// TIA Portal project "Automated Ware house" (V14)
// Vorlageprojekt für das Buch mit Zielsystem S7-1200

(* hardware
DEVICE "S7-1200-Station_1"  S7-1200 Station
   slot 0: "Baugruppenträger_0"  Rack  V1.0
   slot 1: "PLC_1"  CPU 1211C DC/DC/DC  6ES7 211-1AE40-0XB0  V4.1
*)

// ===== PLC "PLC_1"  CPU 1211C DC/DC/DC =====

VAR_GLOBAL   // PLC tag table "Standard-Variablentabelle"
   "At entry" AT %I0.0 : Bool;
   "at load" AT %I0.1 : Bool;
   "at left" AT %I0.2 : Bool;
   "at middle" AT %I0.3 : Bool;
   "at right" AT %I0.4 : Bool;
   "at unload" AT %I0.5 : Bool;
   "at exit" AT %I0.6 : Bool;
   "moving x" AT %I0.7 : Bool;
   "moving z" AT %I1.0 : Bool;
   "start" AT %I1.1 : Bool;
   "reset" AT %I1.2 : Bool;
   "stop" AT %I1.3 : Bool;
   "emergency stop" AT %I1.4 : Bool;
   "auto" AT %I1.5 : Bool;
   "entry conveyor" AT %Q0.0 : Bool;
   "load conveyor" AT %Q0.1 : Bool;
   "forks left" AT %Q0.2 : Bool;
   "fork right" AT %Q0.3 : Bool;
   "lift" AT %Q0.4 : Bool;
   "unload conveyor" AT %Q0.5 : Bool;
   "exit conveyor" AT %Q0.6 : Bool;
   "start light" AT %Q0.7 : Bool;
   "reset light" AT %Q1.0 : Bool;
   "stop light" AT %Q1.1 : Bool;
   "target position" AT %QD30 : DInt;
   "Tag_1" AT %M20.0 : Bool;
   "Tag_2" AT %M20.1 : Bool;
   "Tag_4" AT %MD4 : DInt;
   "Tag_7" AT %MD12 : DInt;
   "Tag_8" AT %M20.2 : Bool;
   "Tag_3" AT %M20.3 : Bool;
   "Tag_14" AT %M21.2 : Bool;
   "Tag_16" AT %M21.4 : Bool;
   "Tag_18" AT %MD8 : DInt;
   "Tag_6" AT %M21.6 : Bool;
   "Tag_19" AT %M21.7 : Bool;
   "Tag_20" AT %M22.1 : Bool;
   "Tag_22" AT %M22.3 : Bool;
   "Tag_5" AT %M22.2 : Bool;
END_VAR

// folder: System blocks/Program resources

DATA_BLOCK "IEC_Counter_0_DB"   // DB1
{ S7_Optimized_Access := 'TRUE' }
AUTHOR : Simatic
FAMILY : IEC
NAME : CNTR
VERSION : 1.0
// stored: InstanceOfName IEC_COUNTER
"IEC_COUNTER"
BEGIN
END_DATA_BLOCK

DATA_BLOCK "IEC_Timer_0_DB"   // DB2
{ S7_Optimized_Access := 'TRUE' }
AUTHOR : Simatic
FAMILY : IEC
NAME : IEC_TMR
VERSION : 1.0
// stored: InstanceOfName IEC_TIMER
"IEC_TIMER"
BEGIN
END_DATA_BLOCK

// folder: (top level)

FUNCTION "Conveyors" : Void   // FC1, LAD
{ S7_Optimized_Access := 'TRUE' }
VERSION : 0.1
   VAR_TEMP   // added for the SCL form of the ladder/FBD networks
      _w1 : Bool;
   END_VAR
BEGIN

REGION Network 1
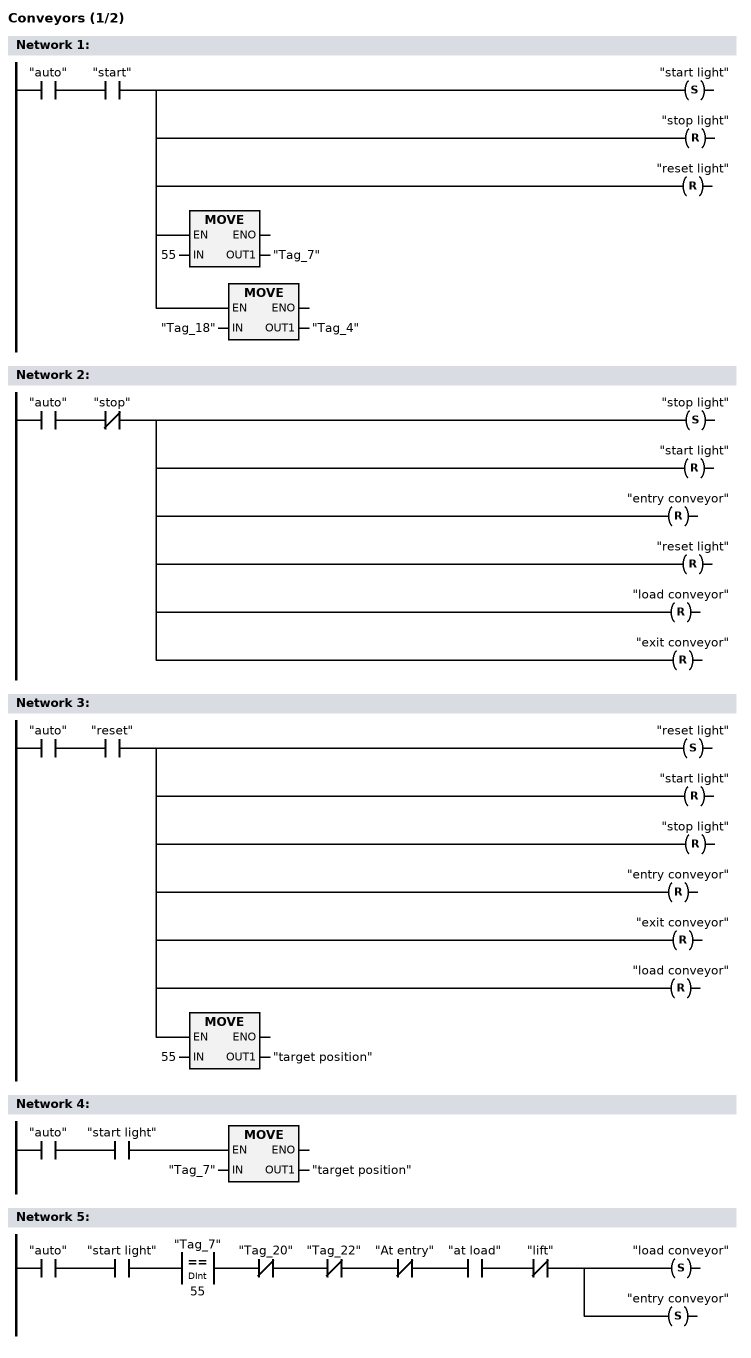
   RUNG wire#powerrail
      Contact( "auto" )
      Contact( "start" )
      wire#w1
      S_Coil( "start light" )
   END_RUNG
   RUNG wire#w1
      R_Coil( "stop light" )
   END_RUNG
   RUNG wire#w1
      R_Coil( "reset light" )
   END_RUNG
   RUNG wire#w1
      Move(in := 55, out1 => "Tag_7")
   END_RUNG
   RUNG wire#w1
      Move(in := "Tag_18", out1 => "Tag_4")
   END_RUNG
   // the same network as SCL:
   IF "auto" AND "start" THEN
       "start light" := TRUE;
       "stop light" := FALSE;
       "reset light" := FALSE;
       "Tag_7" := 55;
       "Tag_4" := "Tag_18";
   END_IF;
END_REGION

REGION Network 2
   RUNG wire#powerrail
      Contact( "auto" )
      I_Contact( "stop" )
      wire#w1
      S_Coil( "stop light" )
   END_RUNG
   RUNG wire#w1
      R_Coil( "start light" )
   END_RUNG
   RUNG wire#w1
      R_Coil( "entry conveyor" )
   END_RUNG
   RUNG wire#w1
      R_Coil( "reset light" )
   END_RUNG
   RUNG wire#w1
      R_Coil( "load conveyor" )
   END_RUNG
   RUNG wire#w1
      R_Coil( "exit conveyor" )
   END_RUNG
   // the same network as SCL:
   IF "auto" AND NOT "stop" THEN
       "stop light" := TRUE;
       "start light" := FALSE;
       "entry conveyor" := FALSE;
       "reset light" := FALSE;
       "load conveyor" := FALSE;
       "exit conveyor" := FALSE;
   END_IF;
END_REGION

REGION Network 3
   RUNG wire#powerrail
      Contact( "auto" )
      Contact( "reset" )
      wire#w1
      S_Coil( "reset light" )
   END_RUNG
   RUNG wire#w1
      R_Coil( "start light" )
   END_RUNG
   RUNG wire#w1
      R_Coil( "stop light" )
   END_RUNG
   RUNG wire#w1
      R_Coil( "entry conveyor" )
   END_RUNG
   RUNG wire#w1
      R_Coil( "exit conveyor" )
   END_RUNG
   RUNG wire#w1
      R_Coil( "load conveyor" )
   END_RUNG
   RUNG wire#w1
      Move(in := 55, out1 => "target position")
   END_RUNG
   // the same network as SCL:
   IF "auto" AND "reset" THEN
       "reset light" := TRUE;
       "start light" := FALSE;
       "stop light" := FALSE;
       "entry conveyor" := FALSE;
       "exit conveyor" := FALSE;
       "load conveyor" := FALSE;
       "target position" := 55;
   END_IF;
END_REGION

REGION Network 4
   RUNG wire#powerrail
      Contact( "auto" )
      Contact( "start light" )
      Move(in := "Tag_7", out1 => "target position")
   END_RUNG
   // the same network as SCL:
   IF "auto" AND "start light" THEN "target position" := "Tag_7"; END_IF;
END_REGION

REGION Network 5
   RUNG wire#powerrail
      Contact( "auto" )
      Contact( "start light" )
      { S7_Templates := "SrcType := DInt" } EQ_Contact(in1 := "Tag_7", in2 := 55)
      I_Contact( "Tag_20" )
      I_Contact( "Tag_22" )
      I_Contact( "At entry" )
      Contact( "at load" )
      I_Contact( "lift" )
      wire#w1
      S_Coil( "load conveyor" )
   END_RUNG
   RUNG wire#w1
      S_Coil( "entry conveyor" )
   END_RUNG
   // the same network as SCL:
   IF "auto" AND "start light" AND ("Tag_7" = 55) AND NOT "Tag_20" AND NOT "Tag_22" AND NOT "At entry" AND "at load" AND NOT "lift" THEN
       "load conveyor" := TRUE;
       "entry conveyor" := TRUE;
   END_IF;
END_REGION

REGION Network 6
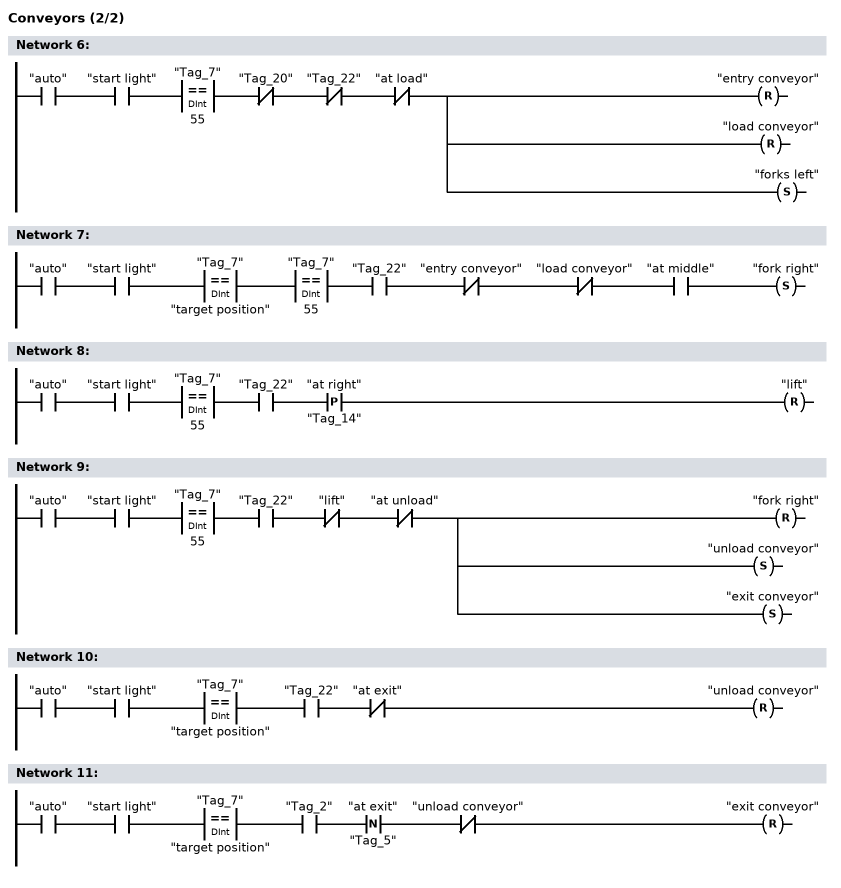
   RUNG wire#powerrail
      Contact( "auto" )
      Contact( "start light" )
      { S7_Templates := "SrcType := DInt" } EQ_Contact(in1 := "Tag_7", in2 := 55)
      I_Contact( "Tag_20" )
      I_Contact( "Tag_22" )
      I_Contact( "at load" )
      wire#w1
      R_Coil( "entry conveyor" )
   END_RUNG
   RUNG wire#w1
      R_Coil( "load conveyor" )
   END_RUNG
   RUNG wire#w1
      S_Coil( "forks left" )
   END_RUNG
   // the same network as SCL:
   IF "auto" AND "start light" AND ("Tag_7" = 55) AND NOT "Tag_20" AND NOT "Tag_22" AND NOT "at load" THEN
       "entry conveyor" := FALSE;
       "load conveyor" := FALSE;
       "forks left" := TRUE;
   END_IF;
END_REGION

REGION Network 7
   RUNG wire#powerrail
      Contact( "auto" )
      Contact( "start light" )
      { S7_Templates := "SrcType := DInt" } EQ_Contact(in1 := "Tag_7", in2 := "target position")
      { S7_Templates := "SrcType := DInt" } EQ_Contact(in1 := "Tag_7", in2 := 55)
      Contact( "Tag_22" )
      I_Contact( "entry conveyor" )
      I_Contact( "load conveyor" )
      Contact( "at middle" )
      S_Coil( "fork right" )
   END_RUNG
   // the same network as SCL:
   IF "auto" AND "start light" AND ("Tag_7" = "target position") AND ("Tag_7" = 55) AND "Tag_22" AND NOT "entry conveyor" AND NOT "load conveyor" AND "at middle" THEN
       "fork right" := TRUE;
   END_IF;
END_REGION

REGION Network 8
   RUNG wire#powerrail
      Contact( "auto" )
      Contact( "start light" )
      { S7_Templates := "SrcType := DInt" } EQ_Contact(in1 := "Tag_7", in2 := 55)
      Contact( "Tag_22" )
      P_Contact(operand := "at right", bit := "Tag_14")
      R_Coil( "lift" )
   END_RUNG
   // the same network as SCL:
   #_w1 := "auto" AND "start light" AND ("Tag_7" = 55) AND "Tag_22" AND "at right" AND NOT "Tag_14";   // rising edge of "at right"
   "Tag_14" := "at right";
   IF #_w1 THEN "lift" := FALSE; END_IF;
END_REGION

REGION Network 9
   RUNG wire#powerrail
      Contact( "auto" )
      Contact( "start light" )
      { S7_Templates := "SrcType := DInt" } EQ_Contact(in1 := "Tag_7", in2 := 55)
      Contact( "Tag_22" )
      I_Contact( "lift" )
      I_Contact( "at unload" )
      wire#w1
      R_Coil( "fork right" )
   END_RUNG
   RUNG wire#w1
      S_Coil( "unload conveyor" )
   END_RUNG
   RUNG wire#w1
      S_Coil( "exit conveyor" )
   END_RUNG
   // the same network as SCL:
   IF "auto" AND "start light" AND ("Tag_7" = 55) AND "Tag_22" AND NOT "lift" AND NOT "at unload" THEN
       "fork right" := FALSE;
       "unload conveyor" := TRUE;
       "exit conveyor" := TRUE;
   END_IF;
END_REGION

REGION Network 10
   RUNG wire#powerrail
      Contact( "auto" )
      Contact( "start light" )
      { S7_Templates := "SrcType := DInt" } EQ_Contact(in1 := "Tag_7", in2 := "target position")
      Contact( "Tag_22" )
      I_Contact( "at exit" )
      R_Coil( "unload conveyor" )
   END_RUNG
   // the same network as SCL:
   IF "auto" AND "start light" AND ("Tag_7" = "target position") AND "Tag_22" AND NOT "at exit" THEN
       "unload conveyor" := FALSE;
   END_IF;
END_REGION

REGION Network 11
   RUNG wire#powerrail
      Contact( "auto" )
      Contact( "start light" )
      { S7_Templates := "SrcType := DInt" } EQ_Contact(in1 := "Tag_7", in2 := "target position")
      Contact( "Tag_2" )
      N_Contact(operand := "at exit", bit := "Tag_5")
      I_Contact( "unload conveyor" )
      R_Coil( "exit conveyor" )
   END_RUNG
   // the same network as SCL:
   #_w1 := "auto" AND "start light" AND ("Tag_7" = "target position") AND "Tag_2" AND NOT "at exit" AND "Tag_5";   // falling edge of "at exit"
   "Tag_5" := "at exit";
   IF #_w1 AND NOT "unload conveyor" THEN "exit conveyor" := FALSE; END_IF;
END_REGION
END_FUNCTION

FUNCTION "Shifting" : Void   // FC2, LAD
{ S7_Optimized_Access := 'TRUE' }
VERSION : 0.1
   VAR_TEMP   // added for the SCL form of the ladder/FBD networks
      _w1 : Bool;
   END_VAR
BEGIN

REGION Network 1
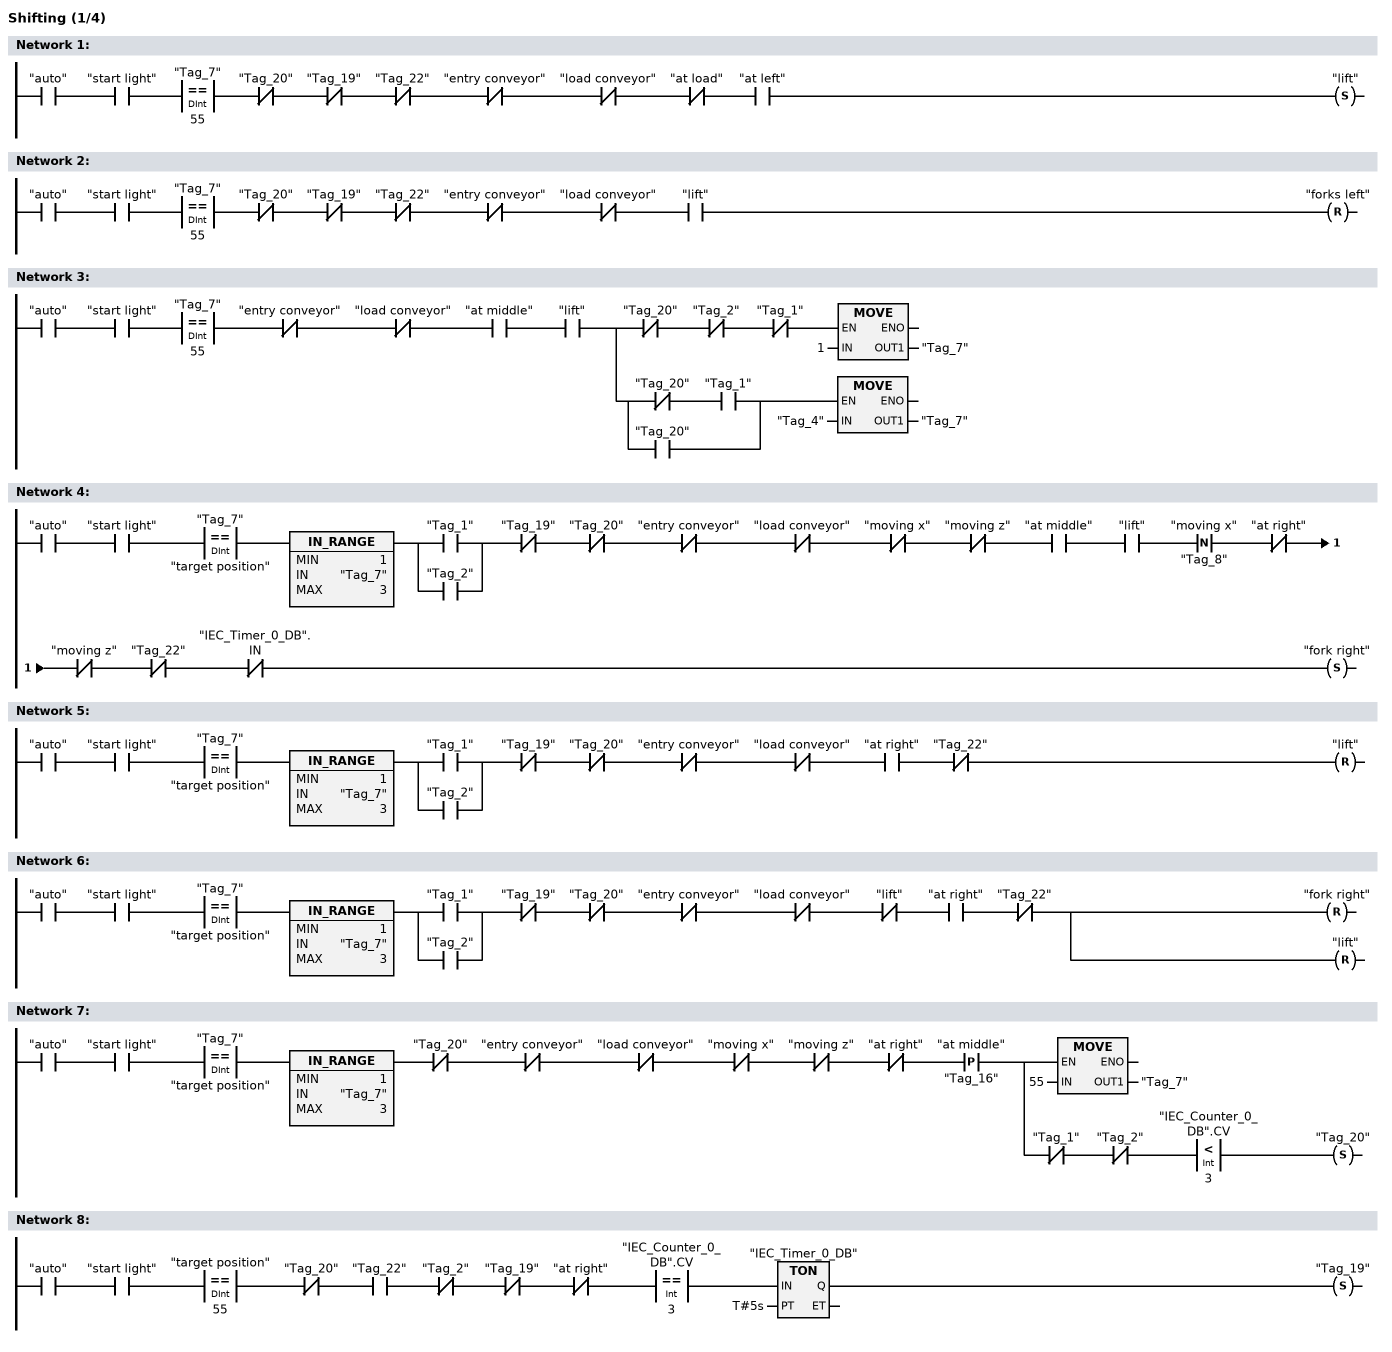
   RUNG wire#powerrail
      Contact( "auto" )
      Contact( "start light" )
      { S7_Templates := "SrcType := DInt" } EQ_Contact(in1 := "Tag_7", in2 := 55)
      I_Contact( "Tag_20" )
      I_Contact( "Tag_19" )
      I_Contact( "Tag_22" )
      I_Contact( "entry conveyor" )
      I_Contact( "load conveyor" )
      I_Contact( "at load" )
      Contact( "at left" )
      S_Coil( "lift" )
   END_RUNG
   // the same network as SCL:
   IF "auto" AND "start light" AND ("Tag_7" = 55) AND NOT "Tag_20" AND NOT "Tag_19" AND NOT "Tag_22" AND NOT "entry conveyor" AND NOT "load conveyor" AND NOT "at load" AND "at left" THEN
       "lift" := TRUE;
   END_IF;
END_REGION

REGION Network 2
   RUNG wire#powerrail
      Contact( "auto" )
      Contact( "start light" )
      { S7_Templates := "SrcType := DInt" } EQ_Contact(in1 := "Tag_7", in2 := 55)
      I_Contact( "Tag_20" )
      I_Contact( "Tag_19" )
      I_Contact( "Tag_22" )
      I_Contact( "entry conveyor" )
      I_Contact( "load conveyor" )
      Contact( "lift" )
      R_Coil( "forks left" )
   END_RUNG
   // the same network as SCL:
   IF "auto" AND "start light" AND ("Tag_7" = 55) AND NOT "Tag_20" AND NOT "Tag_19" AND NOT "Tag_22" AND NOT "entry conveyor" AND NOT "load conveyor" AND "lift" THEN
       "forks left" := FALSE;
   END_IF;
END_REGION

REGION Network 3
   RUNG wire#powerrail
      Contact( "auto" )
      Contact( "start light" )
      { S7_Templates := "SrcType := DInt" } EQ_Contact(in1 := "Tag_7", in2 := 55)
      I_Contact( "entry conveyor" )
      I_Contact( "load conveyor" )
      Contact( "at middle" )
      Contact( "lift" )
      wire#w1
      I_Contact( "Tag_20" )
      I_Contact( "Tag_2" )
      I_Contact( "Tag_1" )
      Move(in := 1, out1 => "Tag_7")
   END_RUNG
   RUNG wire#w1
      I_Contact( "Tag_20" )
      Contact( "Tag_1" )
      wire#w2
      Move(in := "Tag_4", out1 => "Tag_7")
   END_RUNG
   RUNG wire#w1
      Contact( "Tag_20" )
   END_RUNG wire#w2
   // the same network as SCL:
   #_w1 := "auto" AND "start light" AND ("Tag_7" = 55) AND NOT "entry conveyor" AND NOT "load conveyor" AND "at middle" AND "lift";
   IF #_w1 AND NOT "Tag_20" AND NOT "Tag_2" AND NOT "Tag_1" THEN "Tag_7" := 1; END_IF;
   IF #_w1 AND ((NOT "Tag_20" AND "Tag_1") OR "Tag_20") THEN "Tag_7" := "Tag_4"; END_IF;
END_REGION

REGION Network 4
   RUNG wire#powerrail
      Contact( "auto" )
      Contact( "start light" )
      { S7_Templates := "SrcType := DInt" } EQ_Contact(in1 := "Tag_7", in2 := "target position")
      { S7_Templates := "SrcType := DInt" } InRange(min := 1, in := "Tag_7", max := 3)
      wire#w1
      Contact( "Tag_1" )
      wire#w2
      I_Contact( "Tag_19" )
      I_Contact( "Tag_20" )
      I_Contact( "entry conveyor" )
      I_Contact( "load conveyor" )
      I_Contact( "moving x" )
      I_Contact( "moving z" )
      Contact( "at middle" )
      Contact( "lift" )
      N_Contact(operand := "moving x", bit := "Tag_8")
      I_Contact( "at right" )
      I_Contact( "moving z" )
      I_Contact( "Tag_22" )
      I_Contact( "IEC_Timer_0_DB".IN )
      S_Coil( "fork right" )
   END_RUNG
   RUNG wire#w1
      Contact( "Tag_2" )
   END_RUNG wire#w2
   // the same network as SCL:
   #_w1 := "auto" AND "start light" AND ("Tag_7" = "target position") AND (1 <= "Tag_7") AND ("Tag_7" <= 3) AND ("Tag_1" OR "Tag_2") AND NOT "Tag_19" AND NOT "Tag_20" AND NOT "entry conveyor" AND NOT "load conveyor" AND NOT "moving x" AND NOT "moving z" AND "at middle" AND "lift" AND NOT "moving x" AND "Tag_8";   // falling edge of "moving x"
   "Tag_8" := "moving x";
   IF #_w1 AND NOT "at right" AND NOT "moving z" AND NOT "Tag_22" AND NOT "IEC_Timer_0_DB".IN THEN
       "fork right" := TRUE;
   END_IF;
END_REGION

REGION Network 5
   RUNG wire#powerrail
      Contact( "auto" )
      Contact( "start light" )
      { S7_Templates := "SrcType := DInt" } EQ_Contact(in1 := "Tag_7", in2 := "target position")
      { S7_Templates := "SrcType := DInt" } InRange(min := 1, in := "Tag_7", max := 3)
      wire#w1
      Contact( "Tag_1" )
      wire#w2
      I_Contact( "Tag_19" )
      I_Contact( "Tag_20" )
      I_Contact( "entry conveyor" )
      I_Contact( "load conveyor" )
      Contact( "at right" )
      I_Contact( "Tag_22" )
      R_Coil( "lift" )
   END_RUNG
   RUNG wire#w1
      Contact( "Tag_2" )
   END_RUNG wire#w2
   // the same network as SCL:
   IF "auto" AND "start light" AND ("Tag_7" = "target position") AND (1 <= "Tag_7") AND ("Tag_7" <= 3) AND ("Tag_1" OR "Tag_2") AND NOT "Tag_19" AND NOT "Tag_20" AND NOT "entry conveyor" AND NOT "load conveyor" AND "at right" AND NOT "Tag_22" THEN
       "lift" := FALSE;
   END_IF;
END_REGION

REGION Network 6
   RUNG wire#powerrail
      Contact( "auto" )
      Contact( "start light" )
      { S7_Templates := "SrcType := DInt" } EQ_Contact(in1 := "Tag_7", in2 := "target position")
      { S7_Templates := "SrcType := DInt" } InRange(min := 1, in := "Tag_7", max := 3)
      wire#w1
      Contact( "Tag_1" )
      wire#w2
      I_Contact( "Tag_19" )
      I_Contact( "Tag_20" )
      I_Contact( "entry conveyor" )
      I_Contact( "load conveyor" )
      I_Contact( "lift" )
      Contact( "at right" )
      I_Contact( "Tag_22" )
      wire#w3
      R_Coil( "fork right" )
   END_RUNG
   RUNG wire#w1
      Contact( "Tag_2" )
   END_RUNG wire#w2
   RUNG wire#w3
      R_Coil( "lift" )
   END_RUNG
   // the same network as SCL:
   IF "auto" AND "start light" AND ("Tag_7" = "target position") AND (1 <= "Tag_7") AND ("Tag_7" <= 3) AND ("Tag_1" OR "Tag_2") AND NOT "Tag_19" AND NOT "Tag_20" AND NOT "entry conveyor" AND NOT "load conveyor" AND NOT "lift" AND "at right" AND NOT "Tag_22" THEN
       "fork right" := FALSE;
       "lift" := FALSE;
   END_IF;
END_REGION

REGION Network 7
   RUNG wire#powerrail
      Contact( "auto" )
      Contact( "start light" )
      { S7_Templates := "SrcType := DInt" } EQ_Contact(in1 := "Tag_7", in2 := "target position")
      { S7_Templates := "SrcType := DInt" } InRange(min := 1, in := "Tag_7", max := 3)
      I_Contact( "Tag_20" )
      I_Contact( "entry conveyor" )
      I_Contact( "load conveyor" )
      I_Contact( "moving x" )
      I_Contact( "moving z" )
      I_Contact( "at right" )
      P_Contact(operand := "at middle", bit := "Tag_16")
      wire#w1
      Move(in := 55, out1 => "Tag_7")
   END_RUNG
   RUNG wire#w1
      I_Contact( "Tag_1" )
      I_Contact( "Tag_2" )
      { S7_Templates := "SrcType := Int" } LT_Contact(in1 := "IEC_Counter_0_DB".CV, in2 := 3)
      S_Coil( "Tag_20" )
   END_RUNG
   // the same network as SCL:
   #_w1 := "auto" AND "start light" AND ("Tag_7" = "target position") AND (1 <= "Tag_7") AND ("Tag_7" <= 3) AND NOT "Tag_20" AND NOT "entry conveyor" AND NOT "load conveyor" AND NOT "moving x" AND NOT "moving z" AND NOT "at right" AND "at middle" AND NOT "Tag_16";   // rising edge of "at middle"
   "Tag_16" := "at middle";
   IF #_w1 THEN "Tag_7" := 55; END_IF;
   IF #_w1 AND NOT "Tag_1" AND NOT "Tag_2" AND ("IEC_Counter_0_DB".CV < 3) THEN "Tag_20" := TRUE; END_IF;
END_REGION

REGION Network 8
   "IEC_Timer_0_DB".TON(IN := "auto" AND "start light" AND ("target position" = 55) AND NOT "Tag_20" AND "Tag_22" AND NOT "Tag_2" AND NOT "Tag_19" AND NOT "at right" AND ("IEC_Counter_0_DB".CV = 3),
                        PT := T#5s);
   IF "IEC_Timer_0_DB".Q THEN "Tag_19" := TRUE; END_IF;
END_REGION

REGION Network 9
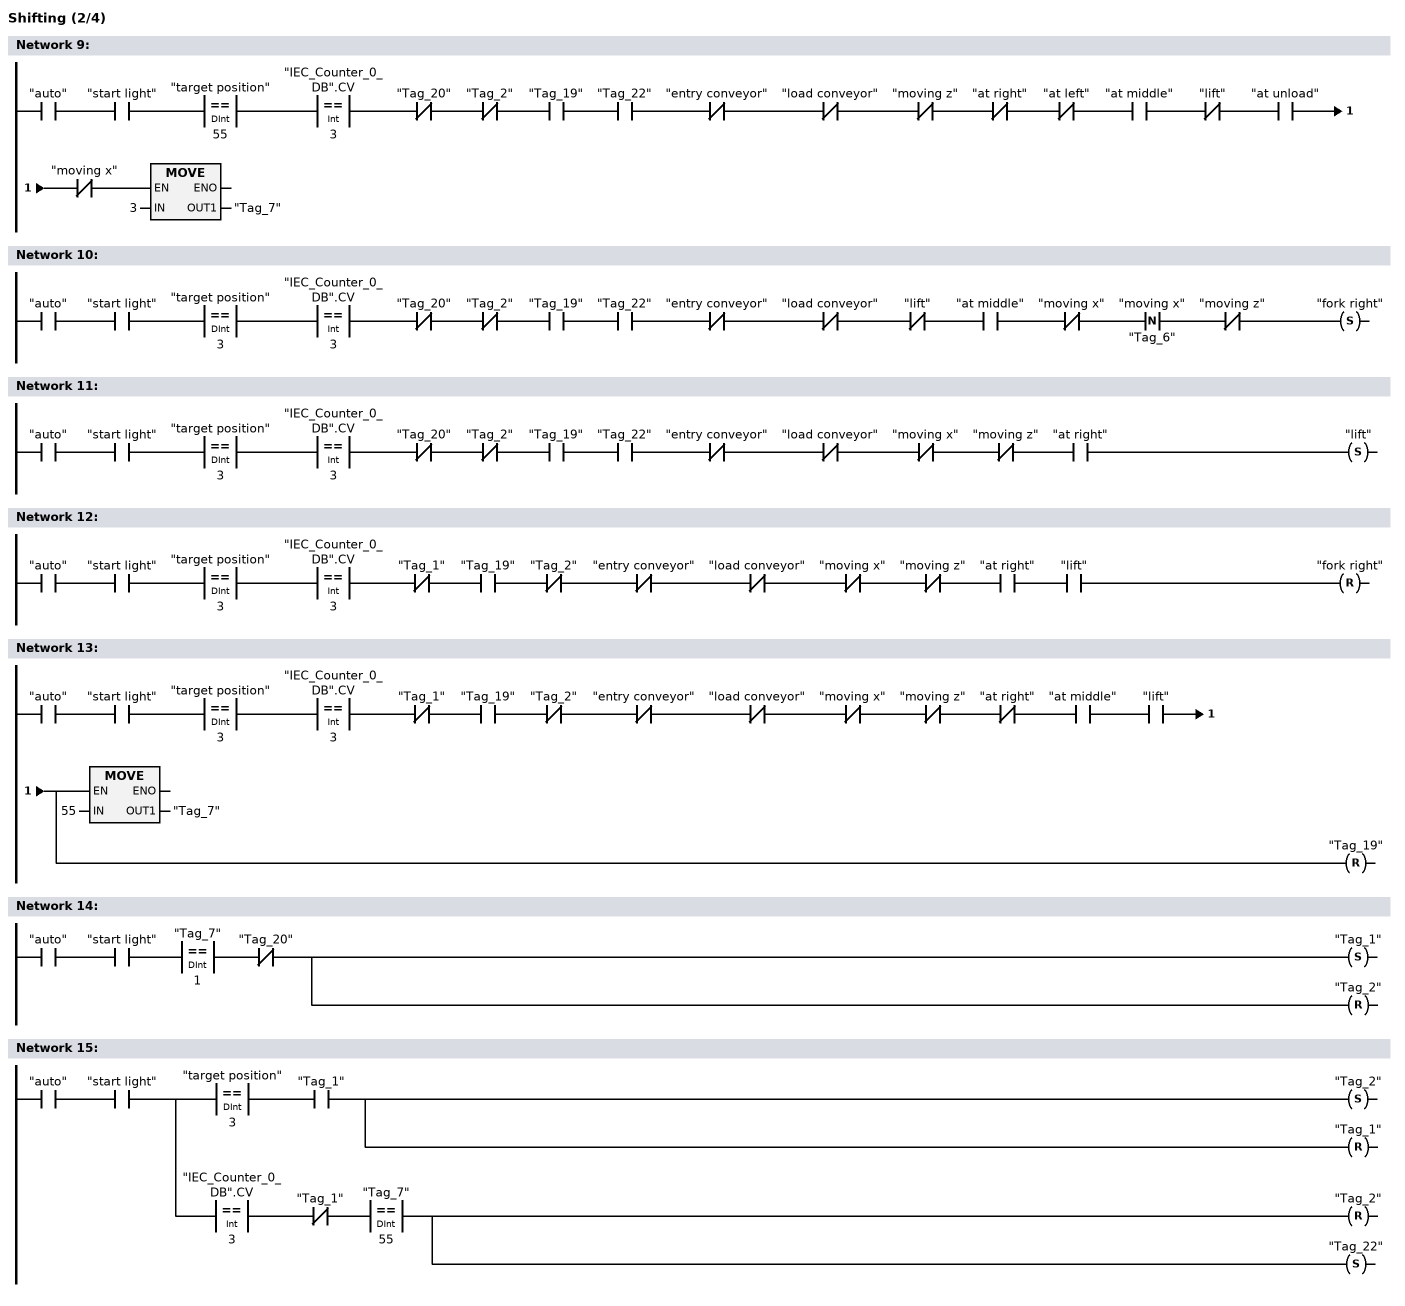
   RUNG wire#powerrail
      Contact( "auto" )
      Contact( "start light" )
      { S7_Templates := "SrcType := DInt" } EQ_Contact(in1 := "target position", in2 := 55)
      { S7_Templates := "SrcType := Int" } EQ_Contact(in1 := "IEC_Counter_0_DB".CV, in2 := 3)
      I_Contact( "Tag_20" )
      I_Contact( "Tag_2" )
      Contact( "Tag_19" )
      Contact( "Tag_22" )
      I_Contact( "entry conveyor" )
      I_Contact( "load conveyor" )
      I_Contact( "moving z" )
      I_Contact( "at right" )
      I_Contact( "at left" )
      Contact( "at middle" )
      I_Contact( "lift" )
      Contact( "at unload" )
      I_Contact( "moving x" )
      Move(in := 3, out1 => "Tag_7")
   END_RUNG
   // the same network as SCL:
   IF "auto" AND "start light" AND ("target position" = 55) AND ("IEC_Counter_0_DB".CV = 3) AND NOT "Tag_20" AND NOT "Tag_2" AND "Tag_19" AND "Tag_22" AND NOT "entry conveyor" AND NOT "load conveyor" AND NOT "moving z" AND NOT "at right" AND NOT "at left" AND "at middle" AND NOT "lift" AND "at unload" AND NOT "moving x" THEN
       "Tag_7" := 3;
   END_IF;
END_REGION

REGION Network 10
   RUNG wire#powerrail
      Contact( "auto" )
      Contact( "start light" )
      { S7_Templates := "SrcType := DInt" } EQ_Contact(in1 := "target position", in2 := 3)
      { S7_Templates := "SrcType := Int" } EQ_Contact(in1 := "IEC_Counter_0_DB".CV, in2 := 3)
      I_Contact( "Tag_20" )
      I_Contact( "Tag_2" )
      Contact( "Tag_19" )
      Contact( "Tag_22" )
      I_Contact( "entry conveyor" )
      I_Contact( "load conveyor" )
      I_Contact( "lift" )
      Contact( "at middle" )
      I_Contact( "moving x" )
      N_Contact(operand := "moving x", bit := "Tag_6")
      I_Contact( "moving z" )
      S_Coil( "fork right" )
   END_RUNG
   // the same network as SCL:
   #_w1 := "auto" AND "start light" AND ("target position" = 3) AND ("IEC_Counter_0_DB".CV = 3) AND NOT "Tag_20" AND NOT "Tag_2" AND "Tag_19" AND "Tag_22" AND NOT "entry conveyor" AND NOT "load conveyor" AND NOT "lift" AND "at middle" AND NOT "moving x" AND NOT "moving x" AND "Tag_6";   // falling edge of "moving x"
   "Tag_6" := "moving x";
   IF #_w1 AND NOT "moving z" THEN "fork right" := TRUE; END_IF;
END_REGION

REGION Network 11
   RUNG wire#powerrail
      Contact( "auto" )
      Contact( "start light" )
      { S7_Templates := "SrcType := DInt" } EQ_Contact(in1 := "target position", in2 := 3)
      { S7_Templates := "SrcType := Int" } EQ_Contact(in1 := "IEC_Counter_0_DB".CV, in2 := 3)
      I_Contact( "Tag_20" )
      I_Contact( "Tag_2" )
      Contact( "Tag_19" )
      Contact( "Tag_22" )
      I_Contact( "entry conveyor" )
      I_Contact( "load conveyor" )
      I_Contact( "moving x" )
      I_Contact( "moving z" )
      Contact( "at right" )
      S_Coil( "lift" )
   END_RUNG
   // the same network as SCL:
   IF "auto" AND "start light" AND ("target position" = 3) AND ("IEC_Counter_0_DB".CV = 3) AND NOT "Tag_20" AND NOT "Tag_2" AND "Tag_19" AND "Tag_22" AND NOT "entry conveyor" AND NOT "load conveyor" AND NOT "moving x" AND NOT "moving z" AND "at right" THEN
       "lift" := TRUE;
   END_IF;
END_REGION

REGION Network 12
   RUNG wire#powerrail
      Contact( "auto" )
      Contact( "start light" )
      { S7_Templates := "SrcType := DInt" } EQ_Contact(in1 := "target position", in2 := 3)
      { S7_Templates := "SrcType := Int" } EQ_Contact(in1 := "IEC_Counter_0_DB".CV, in2 := 3)
      I_Contact( "Tag_1" )
      Contact( "Tag_19" )
      I_Contact( "Tag_2" )
      I_Contact( "entry conveyor" )
      I_Contact( "load conveyor" )
      I_Contact( "moving x" )
      I_Contact( "moving z" )
      Contact( "at right" )
      Contact( "lift" )
      R_Coil( "fork right" )
   END_RUNG
   // the same network as SCL:
   IF "auto" AND "start light" AND ("target position" = 3) AND ("IEC_Counter_0_DB".CV = 3) AND NOT "Tag_1" AND "Tag_19" AND NOT "Tag_2" AND NOT "entry conveyor" AND NOT "load conveyor" AND NOT "moving x" AND NOT "moving z" AND "at right" AND "lift" THEN
       "fork right" := FALSE;
   END_IF;
END_REGION

REGION Network 13
   RUNG wire#powerrail
      Contact( "auto" )
      Contact( "start light" )
      { S7_Templates := "SrcType := DInt" } EQ_Contact(in1 := "target position", in2 := 3)
      { S7_Templates := "SrcType := Int" } EQ_Contact(in1 := "IEC_Counter_0_DB".CV, in2 := 3)
      I_Contact( "Tag_1" )
      Contact( "Tag_19" )
      I_Contact( "Tag_2" )
      I_Contact( "entry conveyor" )
      I_Contact( "load conveyor" )
      I_Contact( "moving x" )
      I_Contact( "moving z" )
      I_Contact( "at right" )
      Contact( "at middle" )
      Contact( "lift" )
      wire#w1
      Move(in := 55, out1 => "Tag_7")
   END_RUNG
   RUNG wire#w1
      R_Coil( "Tag_19" )
   END_RUNG
   // the same network as SCL:
   IF "auto" AND "start light" AND ("target position" = 3) AND ("IEC_Counter_0_DB".CV = 3) AND NOT "Tag_1" AND "Tag_19" AND NOT "Tag_2" AND NOT "entry conveyor" AND NOT "load conveyor" AND NOT "moving x" AND NOT "moving z" AND NOT "at right" AND "at middle" AND "lift" THEN
       "Tag_7" := 55;
       "Tag_19" := FALSE;
   END_IF;
END_REGION

REGION Network 14
   RUNG wire#powerrail
      Contact( "auto" )
      Contact( "start light" )
      { S7_Templates := "SrcType := DInt" } EQ_Contact(in1 := "Tag_7", in2 := 1)
      I_Contact( "Tag_20" )
      wire#w1
      S_Coil( "Tag_1" )
   END_RUNG
   RUNG wire#w1
      R_Coil( "Tag_2" )
   END_RUNG
   // the same network as SCL:
   IF "auto" AND "start light" AND ("Tag_7" = 1) AND NOT "Tag_20" THEN
       "Tag_1" := TRUE;
       "Tag_2" := FALSE;
   END_IF;
END_REGION

REGION Network 15
   RUNG wire#powerrail
      Contact( "auto" )
      Contact( "start light" )
      wire#w1
      { S7_Templates := "SrcType := DInt" } EQ_Contact(in1 := "target position", in2 := 3)
      Contact( "Tag_1" )
      wire#w2
      S_Coil( "Tag_2" )
   END_RUNG
   RUNG wire#w2
      R_Coil( "Tag_1" )
   END_RUNG
   RUNG wire#w1
      { S7_Templates := "SrcType := Int" } EQ_Contact(in1 := "IEC_Counter_0_DB".CV, in2 := 3)
      I_Contact( "Tag_1" )
      { S7_Templates := "SrcType := DInt" } EQ_Contact(in1 := "Tag_7", in2 := 55)
      wire#w3
      R_Coil( "Tag_2" )
   END_RUNG
   RUNG wire#w3
      S_Coil( "Tag_22" )
   END_RUNG
   // the same network as SCL:
   #_w1 := "auto" AND "start light";
   IF #_w1 AND ("target position" = 3) AND "Tag_1" THEN
       "Tag_2" := TRUE;
       "Tag_1" := FALSE;
   END_IF;
   IF #_w1 AND ("IEC_Counter_0_DB".CV = 3) AND NOT "Tag_1" AND ("Tag_7" = 55) THEN
       "Tag_2" := FALSE;
       "Tag_22" := TRUE;
   END_IF;
END_REGION

REGION Network 16
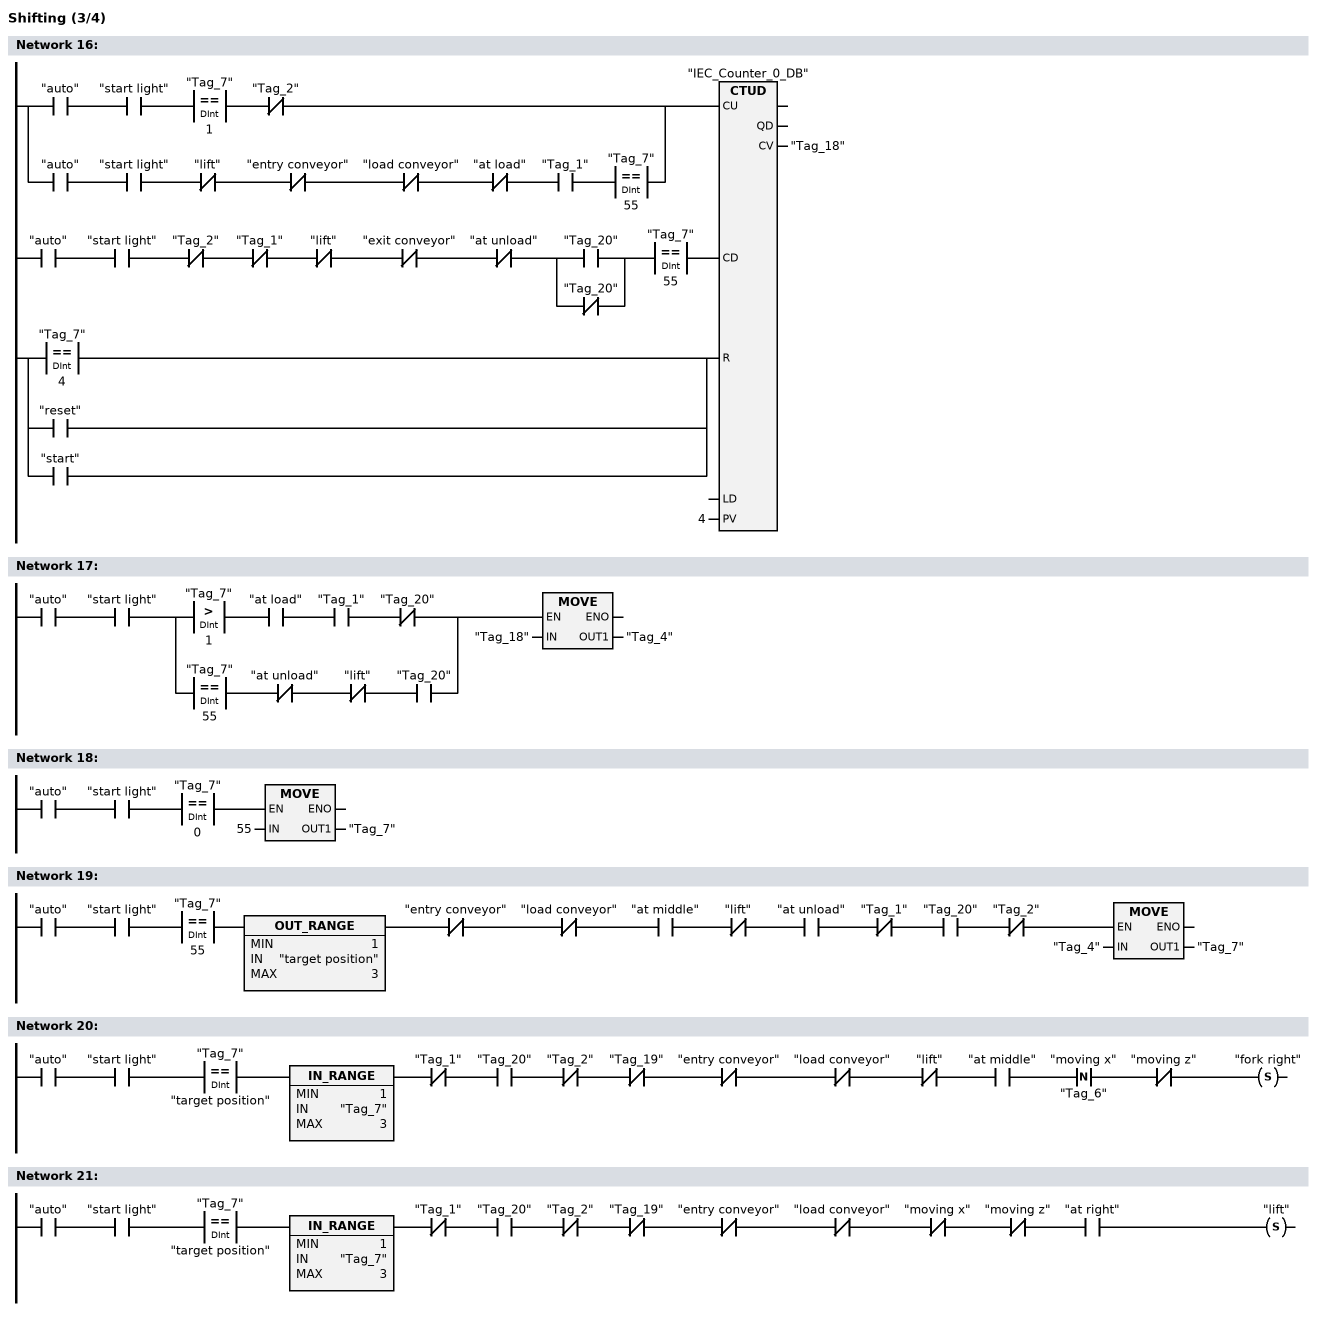
   "IEC_Counter_0_DB".CTUD(CU := ("auto" AND "start light" AND ("Tag_7" = 1) AND NOT "Tag_2") OR ("auto" AND "start light" AND NOT "lift" AND NOT "entry conveyor" AND NOT "load conveyor" AND NOT "at load" AND "Tag_1" AND ("Tag_7" = 55)),
                           CD := "auto" AND "start light" AND NOT "Tag_2" AND NOT "Tag_1" AND NOT "lift" AND NOT "exit conveyor" AND NOT "at unload" AND ("Tag_20" OR NOT "Tag_20") AND ("Tag_7" = 55),
                           R := ("Tag_7" = 4) OR "reset" OR "start",
                           PV := 4,
                           CV => "Tag_18");
END_REGION

REGION Network 17
   RUNG wire#powerrail
      Contact( "auto" )
      Contact( "start light" )
      wire#w1
      { S7_Templates := "SrcType := DInt" } GT_Contact(in1 := "Tag_7", in2 := 1)
      Contact( "at load" )
      Contact( "Tag_1" )
      I_Contact( "Tag_20" )
      wire#w2
      Move(in := "Tag_18", out1 => "Tag_4")
   END_RUNG
   RUNG wire#w1
      { S7_Templates := "SrcType := DInt" } EQ_Contact(in1 := "Tag_7", in2 := 55)
      I_Contact( "at unload" )
      I_Contact( "lift" )
      Contact( "Tag_20" )
   END_RUNG wire#w2
   // the same network as SCL:
   IF "auto" AND "start light" AND ((("Tag_7" > 1) AND "at load" AND "Tag_1" AND NOT "Tag_20") OR (("Tag_7" = 55) AND NOT "at unload" AND NOT "lift" AND "Tag_20")) THEN
       "Tag_4" := "Tag_18";
   END_IF;
END_REGION

REGION Network 18
   RUNG wire#powerrail
      Contact( "auto" )
      Contact( "start light" )
      { S7_Templates := "SrcType := DInt" } EQ_Contact(in1 := "Tag_7", in2 := 0)
      Move(in := 55, out1 => "Tag_7")
   END_RUNG
   // the same network as SCL:
   IF "auto" AND "start light" AND ("Tag_7" = 0) THEN "Tag_7" := 55; END_IF;
END_REGION

REGION Network 19
   IF "auto" AND "start light" AND ("Tag_7" = 55) AND (("target position" < 1) OR ("target position" > 3)) AND NOT "entry conveyor" AND NOT "load conveyor" AND "at middle" AND NOT "lift" AND "at unload" AND NOT "Tag_1" AND "Tag_20" AND NOT "Tag_2" THEN
       "Tag_7" := "Tag_4";
   END_IF;
END_REGION

REGION Network 20
   RUNG wire#powerrail
      Contact( "auto" )
      Contact( "start light" )
      { S7_Templates := "SrcType := DInt" } EQ_Contact(in1 := "Tag_7", in2 := "target position")
      { S7_Templates := "SrcType := DInt" } InRange(min := 1, in := "Tag_7", max := 3)
      I_Contact( "Tag_1" )
      Contact( "Tag_20" )
      I_Contact( "Tag_2" )
      I_Contact( "Tag_19" )
      I_Contact( "entry conveyor" )
      I_Contact( "load conveyor" )
      I_Contact( "lift" )
      Contact( "at middle" )
      N_Contact(operand := "moving x", bit := "Tag_6")
      I_Contact( "moving z" )
      S_Coil( "fork right" )
   END_RUNG
   // the same network as SCL:
   #_w1 := "auto" AND "start light" AND ("Tag_7" = "target position") AND (1 <= "Tag_7") AND ("Tag_7" <= 3) AND NOT "Tag_1" AND "Tag_20" AND NOT "Tag_2" AND NOT "Tag_19" AND NOT "entry conveyor" AND NOT "load conveyor" AND NOT "lift" AND "at middle" AND NOT "moving x" AND "Tag_6";   // falling edge of "moving x"
   "Tag_6" := "moving x";
   IF #_w1 AND NOT "moving z" THEN "fork right" := TRUE; END_IF;
END_REGION

REGION Network 21
   RUNG wire#powerrail
      Contact( "auto" )
      Contact( "start light" )
      { S7_Templates := "SrcType := DInt" } EQ_Contact(in1 := "Tag_7", in2 := "target position")
      { S7_Templates := "SrcType := DInt" } InRange(min := 1, in := "Tag_7", max := 3)
      I_Contact( "Tag_1" )
      Contact( "Tag_20" )
      I_Contact( "Tag_2" )
      I_Contact( "Tag_19" )
      I_Contact( "entry conveyor" )
      I_Contact( "load conveyor" )
      I_Contact( "moving x" )
      I_Contact( "moving z" )
      Contact( "at right" )
      S_Coil( "lift" )
   END_RUNG
   // the same network as SCL:
   IF "auto" AND "start light" AND ("Tag_7" = "target position") AND (1 <= "Tag_7") AND ("Tag_7" <= 3) AND NOT "Tag_1" AND "Tag_20" AND NOT "Tag_2" AND NOT "Tag_19" AND NOT "entry conveyor" AND NOT "load conveyor" AND NOT "moving x" AND NOT "moving z" AND "at right" THEN
       "lift" := TRUE;
   END_IF;
END_REGION

REGION Network 22
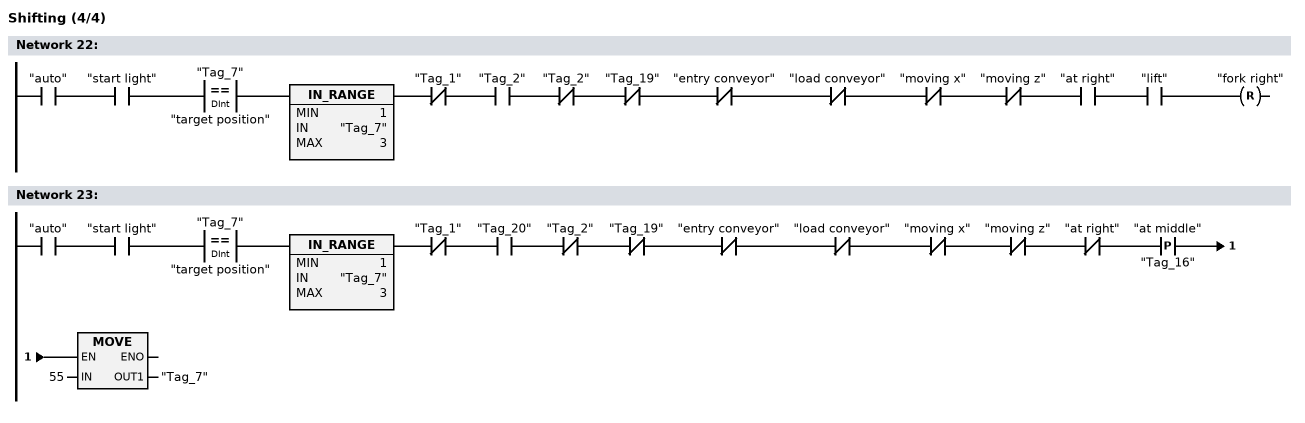
   RUNG wire#powerrail
      Contact( "auto" )
      Contact( "start light" )
      { S7_Templates := "SrcType := DInt" } EQ_Contact(in1 := "Tag_7", in2 := "target position")
      { S7_Templates := "SrcType := DInt" } InRange(min := 1, in := "Tag_7", max := 3)
      I_Contact( "Tag_1" )
      Contact( "Tag_2" )
      I_Contact( "Tag_2" )
      I_Contact( "Tag_19" )
      I_Contact( "entry conveyor" )
      I_Contact( "load conveyor" )
      I_Contact( "moving x" )
      I_Contact( "moving z" )
      Contact( "at right" )
      Contact( "lift" )
      R_Coil( "fork right" )
   END_RUNG
   // the same network as SCL:
   IF "auto" AND "start light" AND ("Tag_7" = "target position") AND (1 <= "Tag_7") AND ("Tag_7" <= 3) AND NOT "Tag_1" AND "Tag_2" AND NOT "Tag_2" AND NOT "Tag_19" AND NOT "entry conveyor" AND NOT "load conveyor" AND NOT "moving x" AND NOT "moving z" AND "at right" AND "lift" THEN
       "fork right" := FALSE;
   END_IF;
END_REGION

REGION Network 23
   RUNG wire#powerrail
      Contact( "auto" )
      Contact( "start light" )
      { S7_Templates := "SrcType := DInt" } EQ_Contact(in1 := "Tag_7", in2 := "target position")
      { S7_Templates := "SrcType := DInt" } InRange(min := 1, in := "Tag_7", max := 3)
      I_Contact( "Tag_1" )
      Contact( "Tag_20" )
      I_Contact( "Tag_2" )
      I_Contact( "Tag_19" )
      I_Contact( "entry conveyor" )
      I_Contact( "load conveyor" )
      I_Contact( "moving x" )
      I_Contact( "moving z" )
      I_Contact( "at right" )
      P_Contact(operand := "at middle", bit := "Tag_16")
      Move(in := 55, out1 => "Tag_7")
   END_RUNG
   // the same network as SCL:
   #_w1 := "auto" AND "start light" AND ("Tag_7" = "target position") AND (1 <= "Tag_7") AND ("Tag_7" <= 3) AND NOT "Tag_1" AND "Tag_20" AND NOT "Tag_2" AND NOT "Tag_19" AND NOT "entry conveyor" AND NOT "load conveyor" AND NOT "moving x" AND NOT "moving z" AND NOT "at right" AND "at middle" AND NOT "Tag_16";   // rising edge of "at middle"
   "Tag_16" := "at middle";
   IF #_w1 THEN "Tag_7" := 55; END_IF;
END_REGION
END_FUNCTION

FUNCTION "MHJ-PLC-Lab-Function-S71200" : Void   // FC9000, SCL
{ S7_Optimized_Access := 'TRUE' }
VERSION : 0.1
   VAR_TEMP
      rdTimeReturn : Int;
      outputTime : DTL;
      SyncVal : Byte;
      forVal : Int;
      forVal_2 : Int;
      Value : Byte;
   END_VAR
   VAR CONSTANT
      CompVal : Byte := 16#34;
      Value_01 : Byte := 16#11;
      Value_01_DW : DWord := 16#A165_D992;
      Value_02_DW : DWord := 16#58BE_4401;
   END_VAR
BEGIN

   #Value:=PEEK(area := 16#82,
        dbNumber := 0,
        byteOffset := 511);
   #Value := #Value + 1;

   POKE(area := 16#82,
        dbNumber := 0,
        byteOffset := 511,
        value := #Value);

   POKE(area:=16#81,
        dbNumber:=0,
        byteOffset:=1016,
        value:=#Value_01_DW);
   POKE(area := 16#81,
        dbNumber := 0,
        byteOffset := 1020,
        value := #Value_02_DW);

   POKE(area := 16#81,
        dbNumber := 0,
        byteOffset := 511,
        value := B#16#00);

   FOR #forVal := 0 TO 120 DO
       FOR #forVal_2:=0 TO 10 DO
           #rdTimeReturn:=RD_SYS_T(#outputTime);
           #rdTimeReturn := WR_SYS_T(#outputTime);
           #rdTimeReturn := RD_SYS_T(#outputTime);
           #rdTimeReturn := WR_SYS_T(#outputTime);
       END_FOR;
       #SyncVal:= PEEK(area := 16#81,
                      dbNumber := 0,
                      byteOffset := 511);
       IF #SyncVal = #CompVal THEN
          GOTO M_1;
       END_IF;
   END_FOR;
   RETURN;

   M_1:
   POKE(area := 16#81,
        dbNumber := 0,
        byteOffset := 511,
        value := B#16#0);
END_FUNCTION

ORGANIZATION_BLOCK "Main"   // OB1, FBD, ProgramCycle
TITLE = "Main Program Sweep (Cycle)"
{ S7_Optimized_Access := 'TRUE' }
VERSION : 0.1
   VAR_INPUT
      Initial_Call : Bool;   // Initial call of this OB
      Remanence : Bool;   // =True, if remanent data are available
   END_VAR
BEGIN

REGION Network 1: Konnektierungsbaustein für PLC-Lab
   // Im Netzwerk 1 wird der Konnektierungsbaustein für PLC-Lab aufgerufen.
   // Dieser Aufruf darf nicht entfernt werden!
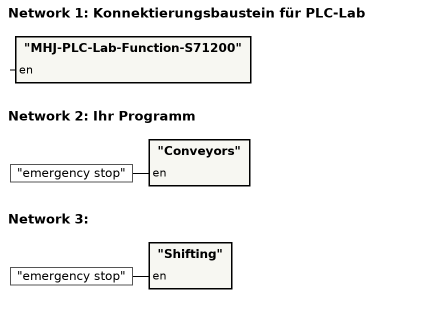
   "MHJ-PLC-Lab-Function-S71200"();
END_REGION

REGION Network 2: Ihr Programm
   // Schreiben Sie ab Netzwerk 2 Ihr Programm
   IF "emergency stop" THEN "Conveyors"(); END_IF;
END_REGION

REGION Network 3
   IF "emergency stop" THEN "Shifting"(); END_IF;
END_REGION
END_ORGANIZATION_BLOCK